# EPICS substitutions: examples/test/el6022/ecmcEL6022_custom.substitutions
file "ecmcEcSlave.template"
{
  pattern {}
          {}
}

file "ecmcEL6022-chX_custom.template"
{
  pattern {CH_ID, NELM }
          {1,     22   }
          {2,     22   }
}
